(* IEC 61131-3 sources: volt/packages/volt-lsp-iec/test-corpus/bakon-nano/Device/Plc Logic/Application/Library Manager/L_EtcSlaveConfig_i700, 25 files *)

(* ---- CHECKVERSION_FIRMWARE_RESULT.dut ---- *)
TYPE CHECKVERSION_FIRMWARE_RESULT :
(
	CVFWR_NO_UPDATE,
	CVFWR_DO_UPDATE,
	CVFWR_HW_INCOMPATIBLE,
	CVFWR_ERROR
);
END_TYPE

(* ---- CHECKVERSION_FIRMWARE_STATE.dut ---- *)
TYPE CHECKVERSION_FIRMWARE_STATE :
(
	CVFW_INITIALIZE,
	CVFW_WAIT_GET_SLAVE_STATE,
	CVFW_SET_SLAVE_STATE_INIT,
	CVFW_SET_SLAVE_STATE_PREOP,
	CVFW_BEFORE_GET_VERSION,
	CVFW_GET_VERSION_I700,
	CVFW_ERROR,
	CVFW_DONE
);
END_TYPE

(* ---- CHECKVERSION_PARAUPLOAD_STATE.dut ---- *)
TYPE CHECKVERSION_PARAUPLOAD_STATE :
(
	CVUP_INITIALIZE,
	CVUP_CHECK_SLAVE_STATE,
	CVUP_GET_FILE_SIZE,
	CVUP_FILE_OPEN,
	CVUP_GET_BUFFER_INDEX,
	CVUP_GET_BUFFER_POINTER,
	CVUP_FILE_READ,
	CVUP_CHECK_FOR_SEL_PS,
	CVUP_READ_CHECKSUM_FROM_SLAVE,
	CVUP_FILE_CLOSE,
	CVUP_ERROR,
	CVUP_DONE
);
END_TYPE

(* ---- CHECKVERSION_STATE.dut ---- *)
TYPE CHECKVERSION_STATE :
(
	CV_NONE,
	CV_INITIALIZE,
	CV_WAIT_GET_SLAVE_STATE,
	CV_SET_SLAVE_STATE_PREOP,
	CV_SLAVE_STATE_IS_PREOP,
	CV_WAIT_FILE_SIZE,
	CV_OPEN_FILE,
	CV_WAIT_FILE_OPEN,
	CV_WAIT_FILE_SET_POS,
	CV_WAIT_FILE_READ_SELECTED_PS_HDR,
	CV_FILE_OPEN,
	CV_CLOSE_FILE,
	CV_CHECK_HDR_FOR_SEL_PS,
	CV_GET_VERSION_I700,
	CV_WAIT_CRC_XFER_COMPLETE,
	CV_ERROR,
	CV_DONE
);
END_TYPE

(* ---- DOWNLOAD_FIRMWARE_STATE.dut ---- *)
TYPE DOWNLOAD_FIRMWARE_STATE :
(
	DLFW_INITIALIZE,
	DLFW_WAIT_BOOTSTRAP_STATE,
	DLFW_GETFILENAMEANDPATH,
	DLFW_GETFILESIZE,
	DLFW_OPENFILE,
	DLFW_GETBUFFERINDEX,
	DLFW_GETBUFFER,
	DLFW_READFILE,
	DLFW_CLOSEFILE,
	DLFW_DOWNLOAD,
	DLFW_RELEASEBUFFER,
	DLFW_ERROR,
	DLFW_ERROR_CLOSE_FILE,
	DLFW_DONE
);
END_TYPE

(* ---- DOWNLOAD_SELECTION_OPTIONS.dut ---- *)
TYPE DOWNLOAD_SELECTION_OPTIONS :
(
	DSELOP_NONE := 0,
	DSELOP_PARAMETER := 1,
	DSELOP_CHANGE := 2,
	DSELOP_ALWAYS := 3,
	DSELOP_NEVER := 4
);
END_TYPE

(* ---- DOWNLOAD_STATE.dut ---- *)
TYPE DOWNLOAD_STATE :
(
	DL_NONE,
	DL_INITIALIZE,
	DL_GETBUFFERINDEX,
	DL_BEFORE_DOWNLOAD,
	DL_OPEN_FILE,
	DL_WAIT_FILE_OPEN,
	DL_FILE_OPEN,
	DL_WAIT_FILE_SET_POS,
	DL_WAIT_FILE_READ,
	DL_CLOSE_FILE,
	DL_WAIT_XFER_COMPLETE,
	DL_ERROR,
	DL_READ_ERROR_FILE,
	DF_ANALYZE_ERROR_FILE,
	DL_AFTER_DOWNLOAD,
	DL_DONE
);
END_TYPE

(* ---- FIRMWARE_DL_MODE.dut ---- *)
TYPE FIRMWARE_DL_MODE :
(
	FWDL_MODE_DISABLED := 0,
	FWDL_MODE_MAIN_VERSION_SLAVE_EQUAL_CONFIGURED_VERSION := 1,
	FWDL_MODE_MAIN_VERSION_SLAVE_GREATER_CONFIGURED_VERSION := 2,
	FWDL_MODE_INDIVIDUAL_CONFIG_AT_SLAVE := 3
);
END_TYPE

(* ---- GETCHECKSUM_STATE.dut ---- *)
TYPE GETCHECKSUM_STATE :
(
	GCS_NONE := 0,
	GCS_GETFILENAMEANDPATH,
	GCS_GETFILESIZE,
	GCS_OPENFILE,
	GCS_READFILE,
	GCS_GETCHECKSUM,
	GCS_CLOSEFILE,
	GCS_ERROR,
	GCS_DONE
);
END_TYPE

(* ---- ONLINEPARADOWNLOAD_STATE.dut ---- *)
TYPE ONLINEPARADOWNLOAD_STATE :
(
	OPD_OPENFILE,
	OPD_WAITFOROPENFILEDONE,
	OPD_DOWNLOAD,
	OPD_ERROR,
	OPD_DONE
);
END_TYPE

(* ---- PARAUPLOAD_STATE.dut ---- *)
TYPE PARAUPLOAD_STATE :
(
	UPL_GETBUFFERINDEX,
	UPL_SETUP,
	UPL_UPLOADING,
	UPL_WAIT_FILE_OPEN,
	UPL_WAIT_FILE_READ_FOR_SEL_PS,
	UPL_WAIT_FILE_OPEN_FOR_SEL_PS,
	UPL_WAIT_FILE_CLOSE_AFTER_READ_FOR_SEL_PS,
	UPL_WAIT_FILE_WRITE_HEADER_FOR_SEL_PS,
	UPL_WAIT_FILE_WRITE_FIRST_OTHER_PARAMETER_SETS_FOR_SEL_PS,
	UPL_WAIT_FILE_WRITE_NEW_PARAMETER_SET_FOR_SEL_PS,
	UPL_WAIT_FILE_WRITE_LAST_OTHER_PARAMETER_SETS_FOR_SEL_PS,
	UPL_WAIT_FILE_CLOSE_AFTER_WRITE_FOR_SEL_PS,
	UPL_WAIT_CALCULATE_CHECKSUM_FOR_SEL_PS,
	UPL_WAIT_FILE_DELETE_OLD_FILE_FOR_SEL_PS,
	UPL_WAIT_FILE_RENAME_OLD_FILE_FOR_SEL_PS,
	UPL_WAIT_FILE_WRITE_DONE,
	UPL_WAIT_FILE_CLOSE_DONE,
	UPL_WAIT_READ_CHECKSUM_DONE,
	UPL_ERROR,
	UPL_DONE
);
END_TYPE

(* ---- RESTART_FIRMWARE_STATE.dut ---- *)
TYPE RESTART_FIRMWARE_STATE :
(
	RSFW_INITIALIZE,
	RSFW_WAIT_FOR_SETSTATE_FINISHED,
	RSFW_WAIT_FOR_STATE_RECEIVED,
	RSFW_ERROR,
	RSFW_DONE,
	RSFW_WAITFORRESTARTFINISH,
	RSFW_SETSTATEPREOP
);
END_TYPE

(* ---- GETBOOLEANPROPERTY.pou ---- *)
FUNCTION GETBOOLEANPROPERTY : BOOL
VAR_INPUT
	STKEY : WSTRING;
END_VAR
END_FUNCTION

(* ---- GETCOMPANY.pou ---- *)
FUNCTION GETCOMPANY : WSTRING
END_FUNCTION

(* ---- GETNUMBERPROPERTY.pou ---- *)
FUNCTION GETNUMBERPROPERTY : DINT
VAR_INPUT
	STKEY : WSTRING;
END_VAR
END_FUNCTION

(* ---- GETTEXTPROPERTY.pou ---- *)
FUNCTION GETTEXTPROPERTY : WSTRING
VAR_INPUT
	STKEY : WSTRING;
END_VAR
END_FUNCTION

(* ---- GETTEXTPROPERTY2.pou ---- *)
FUNCTION GETTEXTPROPERTY2 : POINTER TO WSTRING
VAR_INPUT
	STKEY : WSTRING;
END_VAR
END_FUNCTION

(* ---- GETTITLE.pou ---- *)
FUNCTION GETTITLE : WSTRING
END_FUNCTION

(* ---- GETVERSION.pou ---- *)
FUNCTION GETVERSION : VERSION
END_FUNCTION

(* ---- GETVERSIONPROPERTY.pou ---- *)
FUNCTION GETVERSIONPROPERTY : VERSION
VAR_INPUT
	STKEY : WSTRING;
END_VAR
END_FUNCTION

(* ---- ETCCONFIGPARAUPLOAD_I700.pou ---- *)
FUNCTION_BLOCK ETCCONFIGPARAUPLOAD_I700 EXTENDS L_SUDP_UpDownload
VAR
	ECONTROL : L_SUDP_Control;
	BYOLDVALUEOFCONTROLINPUT : BYTE := 16#FF;
	PETCDEV : POINTER TO ETCSlave;
	UPLSTATE : PARAUPLOAD_STATE := PARAUPLOAD_STATE.UPL_GETBUFFERINDEX;
	GETSLAVESTATE : L_ETC_GetSlaveState;
	GETETCMASTERDIAGNOSTIC : L_ETC_GetMasterDiagnostic;
	ELASTERROR : L_SUDP_ErrorCodes;
	PSATTACHEDERRORTXT : POINTER TO STRING;
	XSHOULDUPLOAD : BOOL;
	CVUPLSTATE : CHECKVERSION_PARAUPLOAD_STATE := CHECKVERSION_PARAUPLOAD_STATE.CVUP_INITIALIZE;
	FOPEN : FILE.Open;
	FREAD : FILE.Read;
	FCLOSE : FILE.Close;
	FGETSIZE : FILE.GetSize;
	FDELETE : FILE.Delete;
	FRENAME : File.Rename;
	SFILENAMEANDPATH : STRING(L_SUDP.L_SUDP_MAX_STRING_LENGTH.PATH_AND_FILE_NAME);
	HPARAFILE : CAA.HANDLE;
	SZFILESIZE : CAA.SIZE;
	READCHECKSUM : L_ETC_CoE_SdoRead;
	DWFILECRC : DWORD;
	DWSLAVECRC : DWORD;
	FOEREAD : L_ETC_FoE_Read;
	FWRITE : FILE.Write;
	GETCHECKSUMOFFILE : L_SUDP_GetChecksumFromPRMFile;
	BYPARSETDLMODEFROMPARAMETER : BYTE;
	IGNOREPARSETUL : BOOL;
	SELPSPARAFILEHEAD : L_SUDP_PAR_FILE_HDR_SEL_PS;
	ISSELECTABLEPARAMETERSET : BOOL;
	SELECTEDPARAMETERSETDATAOFFSET : DWORD;
	DWACTIVEPARAMETERSET : DWORD;
	PBYFILEBUFFER : POINTER TO BYTE;
	SNEWFILENAMEANDPATH : STRING(255);
	DWWRITEPART1FROMPOSITIONFORSELPS : DWORD;
	DWWRITEPART1SIZEFORSELPS : DWORD;
	DWWRITEPART2FROMPOSITIONFORSELPS : DWORD;
	DWWRITEPART2SIZEFORSELPS : DWORD;
	CALCULATECHECKSUM : CalculateChecksumFromOpenFile;
	READ_BUFFER_SIZE_SINGLE_PS : WORD := 15000;
	I700_PAR_SET_FILE_WRITE_TIMEOUT : UDINT := 10000;
END_VAR
END_FUNCTION_BLOCK

METHOD CHECKVERSION
END_METHOD

METHOD GETFILENAMEFORFOETRANSFER : CAA_FILENAME
END_METHOD

METHOD INITIALIZE
VAR_INPUT
	PETCREMDEV : POINTER TO L_ETCSlave_i700;
END_VAR
END_METHOD

METHOD PARAUPLOAD
END_METHOD

METHOD READSELPSFILEHEADER
VAR_INPUT
	BYBUFFER : POINTER TO BYTE;
END_VAR
END_METHOD

METHOD RESETALLSIGNALS : BOOL
END_METHOD

METHOD UPDATESELPSHEADER
VAR_INPUT
	SZNEWSIZESLAVEPS : CAA_SIZE;
	DWACTIVEPS : DWORD;
	PDWWRITEPART1FROMPOSITIONFORSELPS : POINTER TO DWORD;
	PDWWRITEPART1SIZEFORSELPS : POINTER TO DWORD;
	PDWWRITEPART2FROMPOSITIONFORSELPS : POINTER TO DWORD;
	PDWWRITEPART2SIZEFORSELPS : POINTER TO DWORD;
END_VAR
END_METHOD

(* ---- ETCCONFIGPARAXFER_I700.pou ---- *)
FUNCTION_BLOCK ETCCONFIGPARAXFER_I700 EXTENDS L_SUDP_UpDownload
VAR_INPUT
	XPREVENTETCOPERATIONALWHENSDOWRITEERROR : BOOL;
END_VAR
VAR
	BYOLDVALUEOFCONTROLINPUT : BYTE := 16#FF;
	DOWNLOADSTATE : DOWNLOAD_STATE := DOWNLOAD_STATE.DL_GETBUFFERINDEX;
	CHECKVERSIONSTATE : CHECKVERSION_STATE := CHECKVERSION_STATE.CV_INITIALIZE;
	ONLINEPARADOWNLOADSTATE : ONLINEPARADOWNLOAD_STATE := ONLINEPARADOWNLOAD_STATE.OPD_OPENFILE;
	PETCDEV : POINTER TO ETCSlave;
	ECONTROL : L_SUDP_Control;
	ELASTERROR : L_SUDP_ErrorCodes;
	PSATTACHEDERRORTXT : POINTER TO STRING;
	SFILENAMEANDPATH : STRING(L_SUDP.L_SUDP_MAX_STRING_LENGTH.PATH_AND_FILE_NAME);
	PDUMMYALIGNMENT1 : POINTER TO BYTE;
	BYIOBUFFER : ARRAY [0..((SIZEOF(L_SUDP_PAR_FILE_HDR_SEL_PS) + SIZEOF(L_SUDP_PAR_DATA_HDR)) - 1)] OF BYTE;
	PFILEHDR : POINTER TO L_SUDP_PAR_FILE_HDR;
	DWPARAFILESZ : DWORD;
	HPARAFILE : CAA.HANDLE;
	FGETFS : FILE.GetSize;
	FOPEN : FILE.Open;
	FREAD : FILE.Read;
	FCLOSE : FILE.Close;
	FSETPOS : FILE.SetPos;
	SDORD : L_ETC_CoE_SdoRead;
	FOEWR : L_ETC_FoE_Write;
	FOERD : L_ETC_FoE_Read;
	GETSLAVESTATE : L_ETC_GetSlaveState;
	SETSLAVESTATE : L_ETC_SetSlaveStateFWDL;
	DWCRC32 : DWORD;
	GETETCMASTERDIAGNOSTIC : L_ETC_GetMasterDiagnostic;
	XISFIRSTDOWNLOADERROR : BOOL;
	PARAFILEHEAD : L_SUDP_PAR_FILE_HDR;
	SELPSPARAFILEHEAD : L_SUDP_PAR_FILE_HDR_SEL_PS;
	ISSELECTABLEPARAMETERSET : BOOL;
	SELECTEDPARAMETERSETDATAOFFSET : DWORD;
	XBEFOREDOWNLOADDONE : BOOL;
	PPARMDAT : POINTER TO L_SUDP_PAR_DATA_HDR;
	PERRORDAT : POINTER TO L_SUDP_PARM_ERROR_CODE;
	DWERRORLISTSIZECOUNTER : DWORD;
	BYPARSETDLMODEFROMPARAMETER : BYTE;
	IGNOREPARSETDL : BOOL;
	PDUMMYALIGNMENT2 : POINTER TO BYTE;
	ABYERRORLIST : ARRAY [0..30000] OF BYTE;
	SDEBUGTEXT_I700 : STRING(200);
END_VAR
END_FUNCTION_BLOCK

METHOD AFTERDOWNLOAD : BOOL
END_METHOD

METHOD BEFOREDOWNLOAD : BOOL
END_METHOD

METHOD BYTEARRAYTODWORDCONV : DWORD
VAR_INPUT
	PABY : POINTER TO BYTE;
END_VAR
END_METHOD

METHOD BYTEARRAYTOWORDCONV : WORD
VAR_INPUT
	PABY : POINTER TO BYTE;
END_VAR
END_METHOD

METHOD CHECKFILETYPE : BOOL
VAR_INPUT
	DWFILETYPE : DWORD;
END_VAR
END_METHOD

METHOD CHECKVERSION
END_METHOD

METHOD CLOSEFILE
END_METHOD

METHOD DOWNLOAD
END_METHOD

METHOD GETERRORFILENAME : STRING
END_METHOD

METHOD GETFILENAMEFORFOETRANSFER : CAA_FILENAME
END_METHOD

METHOD GETTIMEOUTFORFOEWRITE : UDINT
END_METHOD

METHOD INITIALIZE
VAR_INPUT
	PETCREMDEV : POINTER TO L_ETCSlave_i700;
END_VAR
END_METHOD

METHOD ONSLAVEISPREOP : BOOL
END_METHOD

METHOD ONLINEPARADOWNLOAD
END_METHOD

METHOD READDWORD : DWORD
VAR_INPUT
	PBYBUFFER : POINTER TO BYTE;
	DWOFFSET : DWORD;
END_VAR
END_METHOD

METHOD READPARAFILEHEAD
END_METHOD

METHOD READSELPSFILEHEADER
END_METHOD

METHOD RESETALLSIGNALS : BOOL
END_METHOD

METHOD SETCURRENTPS
VAR_INPUT
	PARSETNUMBER : USINT;
END_VAR
END_METHOD

(* ---- ETCFIRMWAREDOWNLOAD_I700.pou ---- *)
FUNCTION_BLOCK ETCFIRMWAREDOWNLOAD_I700 EXTENDS L_SUDP_UpDownload
VAR
	ECONTROL : L_SUDP_Control;
	BYOLDVALUEOFCONTROLINPUT : BYTE := 16#FF;
	ELASTERROR : L_SUDP_ErrorCodes;
	PSATTACHEDERRORTXT : POINTER TO STRING;
	PETCDEV : POINTER TO ETCSlave;
	CHECKVERSIONSTATE : CHECKVERSION_FIRMWARE_STATE := CVFW_INITIALIZE;
	STARGETVERSION : STRING(L_SUDP.L_SUDP_MAX_STRING_LENGTH.DEVICE_FIRMWARE_VERSION_NUMBER);
	SSLAVEVERSION : STRING((L_SUDP.L_SUDP_MAX_STRING_LENGTH.DEVICE_FIRMWARE_VERSION_NUMBER + 20));
	XISTARGETVERSIONEXIST : BOOL := FALSE;
	READSLAVEFIRMWAREVERSION : L_ETC_CoE_SdoRead;
	READSLAVESDOCOUNTER : INT;
	XISERRORBYCHECKVERSION : BOOL := FALSE;
	SBINARYFILENAME : STRING(L_SUDP.L_SUDP_MAX_STRING_LENGTH.FILE_NAME);
	DOWNLOADSTATE : DOWNLOAD_FIRMWARE_STATE := DLFW_INITIALIZE;
	SETSLAVESTATE : L_ETC_SetSlaveStateFWDL;
	FIRMWAREWRITE : L_ETC_FoE_Write;
	GETSLAVESTATE : L_ETC_GetSlaveState;
	FILEOPEN : FILE.Open;
	FILEREAD : FILE.Read;
	FILECLOSE : FILE.Close;
	FILEGETSIZE : FILE.GetSize;
	EREADERROR : FILE.ERROR;
	HFILEHANDLE : CAA.HANDLE;
	EGETBUFFERERROR : L_SUDP_ErrorCodes;
	XDUMMY : BOOL;
	XISNAMEGOT : BOOL;
	SPATHANDNAME : STRING(L_SUDP.L_SUDP_MAX_STRING_LENGTH.PATH_AND_FILE_NAME);
	SZFILESIZE : CAA.SIZE;
	XISFIRSTDOWNLOADERROR : BOOL;
	RESTARTSTATE : RESTART_FIRMWARE_STATE := RSFW_INITIALIZE;
	RESTARTSTATE2 : RESTART_FIRMWARE_STATE := RSFW_INITIALIZE;
	STARTTIME : CAA.TICK;
	ENDTIME : CAA.TICK;
	RESTARTDELAY : Standard.TON;
	GETETCMASTERDIAGNOSTIC : L_ETC_GetMasterDiagnostic;
	WTARGETID : WORD;
	BYFWDLMODEFROMPARAMETER : BYTE;
	IGNOREFWDL : BOOL;
	BTESTONEFIRMWAREDOWNLOADDONE : BOOL;
	NTESTCOUNTER : INT;
	TEST_FW_DOWNLOAD_ACTIVE : BOOL := FALSE;
	TIME_OUT_FW_TRANSFER : UDINT := 40;
	I700_RESTART_TIMEOUT : TIME := TIME#1s500ms;
	MAX_SDO_READ_READ_ATTEMPTS : INT := 11;
END_VAR
END_FUNCTION_BLOCK

METHOD CALLBEFOREGETVERSION
END_METHOD

METHOD CHECKVERSION
END_METHOD

METHOD CLOSEFILE
END_METHOD

METHOD DOWNLOAD
END_METHOD

METHOD GETFILENAMEFORFOETRANSFER : CAA_FILENAME
END_METHOD

METHOD GETTIMEOUTFORFOEFIRMWARETRANSFER : UDINT
END_METHOD

METHOD INITIALIZE
VAR_INPUT
	PETCREMDEV : POINTER TO L_ETCSlave_i700;
END_VAR
END_METHOD

METHOD ISDOWNLOADNECESSARY : CHECKVERSION_FIRMWARE_RESULT
VAR_INPUT
	STARGETVERSION : STRING(L_SUDP.L_SUDP_MAX_STRING_LENGTH.DEVICE_FIRMWARE_VERSION_NUMBER);
	SSLAVEVERSION : STRING((L_SUDP.L_SUDP_MAX_STRING_LENGTH.DEVICE_FIRMWARE_VERSION_NUMBER + 20));
	BYFWDLMODE : BYTE;
END_VAR
END_METHOD

METHOD ISFIRMWAREDOWNLOADTYPE2 : BOOL
VAR_INPUT
	WTARGETID : WORD;
END_VAR
END_METHOD

METHOD ISFIRMWAREDOWNLOADTYPEI750 : BOOL
END_METHOD

METHOD MUSTCALLBEFOREGETVERSION : BOOL
END_METHOD

METHOD RESETALLSIGNALS : BOOL
END_METHOD

METHOD RESTARTTYPE1 : BOOL
END_METHOD

METHOD RESTARTTYPE2_1
END_METHOD

METHOD RESTARTTYPE2_2
END_METHOD

METHOD RESTARTTYPE_I750
END_METHOD

METHOD SHOULDUPDATE : CHECKVERSION_FIRMWARE_RESULT
VAR_INPUT
	STARGETVERSIONMAJOR : STRING(10);
	STARGETVERSIONMINOR : STRING(10);
	STARGETVERSIONPATCHLEVEL : STRING(10);
	STARGETVERSIONBUILDNUMBER : STRING(10);
	SSLAVEVERSIONMAJOR : STRING(10);
	SSLAVEVERSIONMINOR : STRING(10);
	SSLAVEVERSIONPATCHLEVEL : STRING(10);
	SSLAVEVERSIONBUILDNUMBER : STRING(10);
	BYFWDLMODE : BYTE;
END_VAR
END_METHOD

METHOD VERSIONNUMBERANALYSIS : BOOL
VAR_INPUT
	PSVERSION : POINTER TO BYTE;
	PSMAJOR : POINTER TO STRING(10);
	PSMINOR : POINTER TO STRING(10);
	PSPATCHLEVEL : POINTER TO STRING(10);
	PSBUILDNUMBER : POINTER TO STRING(10);
	DWSIZE : DWORD;
END_VAR
END_METHOD

(* ---- L_ETCSLAVE_I700.pou ---- *)
FUNCTION_BLOCK L_ETCSLAVE_I700
VAR_OUTPUT
	PETCSLAVE : POINTER TO ETCSlave;
END_VAR
VAR
	ETCSLAVE : ETCSlave;
	M_HLEMACCESS_I700 : RTS_IEC_HANDLE;
	PARSETXFER : EtcConfigParaXfer_i700;
	FIRMWAREDOWNLOAD : EtcFirmwareDownload_i700;
	PARSETUPLOAD : EtcConfigParaUpload_i700;
	ISMANDATORY : BOOL;
	ISPRESENT : BOOL;
	MODULEHANDLER : L_IMHP_IModuleHandler;
END_VAR
END_FUNCTION_BLOCK

METHOD CYCLICCALL : UDINT
END_METHOD

METHOD FB_EXIT : BOOL
VAR_INPUT
	BINCOPYCODE : BOOL;
END_VAR
END_METHOD

METHOD FB_INIT : BOOL
VAR_INPUT
	BINITRETAINS : BOOL;
	BINCOPYCODE : BOOL;
END_VAR
END_METHOD

METHOD INITIALIZE : UDINT
VAR_INPUT
	WMODULETYPE : UINT;
	DWINSTANCE : UDINT;
	PCONNECTOR : POINTER TO IoConfigConnector;
END_VAR
END_METHOD

(* ---- L_SUDP_GETCHECKSUMFROMPRMFILE.pou ---- *)
FUNCTION_BLOCK L_SUDP_GETCHECKSUMFROMPRMFILE
VAR_INPUT
	XEXECUTE : BOOL;
	EBUSTYPE : L_SUDP_BUS_TYPE;
	WNETID : WORD;
	WSLAVEADR : WORD;
END_VAR
VAR_OUTPUT
	XDONE : BOOL;
	XBUSY : BOOL;
	XERROR : BOOL;
	DWFILECRC : DWORD;
	EERRORCODE : L_SUDP_ErrorCodes := L_SUDP_ErrorCodes.NO_ERROR;
END_VAR
VAR
	SPARAFILEPATH : STRING(200);
	SPARAFILENAME : STRING(120);
	SNETID : STRING(40);
	SPATHANDNAME : STRING(300);
	ESTATE : GETCHECKSUM_STATE := GETCHECKSUM_STATE.GCS_NONE;
	XOLDEXECUTE : BOOL;
	ELASTERROR : L_SUDP_ErrorCodes;
	HFILEHANDLE : CAA.HANDLE;
	SZFILESIZE : CAA.SIZE;
	PFILEHEADER : POINTER TO L_SUDP_PAR_FILE_HDR;
	PPARDATAHEADER : POINTER TO L_SUDP_PAR_DATA_HDR;
	BYIOBUFFER : ARRAY [0..((SIZEOF(L_SUDP_PAR_FILE_HDR) + SIZEOF(L_SUDP_PAR_DATA_HDR)) - 1)] OF BYTE;
	FILEOPEN : FILE.Open;
	FILEREAD : FILE.Read;
	FILECLOSE : FILE.Close;
	FILEGETSIZE : FILE.GetSize;
	FILE_IO_TIMEOUT : UDINT := 10000000;
END_VAR
END_FUNCTION_BLOCK
